(* IEC 61131-3 sources: AXOpen/src/components.siemens.identification/ctrl/src/IOLink, 6 files *)

(* ---- AxoIOLink_Device.st ---- *)
USING AXOpen.Components.Abstractions.Drives;
USING AXOpen.Timers;
USING Siemens.Simatic.S71500.DistributedIO;
USING System.Timer;

NAMESPACE AXOpen.Components.SIEM.Identification
    {S7.extern=ReadWrite}
    CLASS PUBLIC AxoIOLink_Device
        VAR PRIVATE
            statExecuteOld          :	BOOL    :=  FALSE;          //  Old value of 'execute' input for edge detection
            statDone                :	BOOL    :=  FALSE;          //  Static value for output 'done'
            statBusy                :	BOOL    :=  FALSE;          //  Static value for output 'busy'
            statError               :	BOOL    :=  FALSE;          //  Static value for output 'error'
            statStatus              :	WORD    :=  WORD#16#7000;	//  Static value for output 'status'
            statPollingPeriod       :	TIME    :=	T#100MS;        //	Static value for input 'pollingPeriod'
            statHwID                :	WORD    :=  WORD#0;         //  Static value for input 'hwID'
            statHwIDprevious        :	WORD    :=  WORD#0;         //  Static value for input 'hwID' from the previous execute
            statReadWrite           :	BOOL    :=  FALSE;          //  Static value for input 'readWrite'
            statCap                 :	UINT    :=  UINT#0;         //  Static value for input 'cap'
            statTimeout             :	TIME    :=	T#0MS;          //	Static value for input 'timeout'
            statLen                 :	UINT    :=  UINT#0;         //  Length of data to be written to device
            statSubfunctionStatus   :	DWORD   :=  DWORD#0;        //  Status of WRREC/RDREC or error code from IO-Link Master (%W1: IO-Link Master error, %W0: ISDU error)
            statFBErrorState        :	DINT    :=  DINT#0;         //	State in the state machine of the block where the error occurred
            statFBState             :	DINT    :=  DINT#0;         //	State in the state machine of the FB
            statEmptyDiagnostics    :	AxoIOLink_typeDiagnostics;  //  Empty diagnostics information (for initialization purposes only)
            instRdRec               :	ReadRecord;                 //  System function "read data record"
            instWrRec               :	WriteRecord;                //  System function "write data record"
            instPoll                :	Pulse;  		            //  poll rate read data record
            instMonitor             :	OnDelay;                    //  request monitoring time
            statRead                :	ARRAY[0..239] OF BYTE   := [BYTE#16#08,BYTE#16#0,BYTE#16#FE,BYTE#16#4A,236(BYTE#0)];             //  data area for reading data
            statWrite               :	ARRAY[0..239] OF BYTE   := [BYTE#16#08,BYTE#16#0,BYTE#16#FE,BYTE#16#4A,236(BYTE#0)];             //  data area for writing data
            statDiagnostics         :	AxoIOLink_typeDiagnostics;
            statReadLen             :	INT;

        END_VAR

        VAR CONSTANT
            MODE_READ                   :	BOOL    :=	FALSE;              //  Mode to read data
            MODE_WRITE                  :	BOOL    :=	TRUE;               //  Mode to write data
            MAX_PORT                    :	USINT   :=  USINT#63;           //  Max. possible port
            MAX_INDEX                   :	UINT    :=  UINT#32767;         //  Max. possible index
            INDEX_PORT_FUNC             :	UINT    :=  UINT#65535;         //  Index to address port functions
            MAX_SUBINDEX                :	USINT   :=  USINT#255;          //  Max. possible subindex
            MAX_DATA                    :	USINT	:=  USINT#232;          //  Max. size of data to be transferred
            UPPER_LIMIT                 :	DINT    :=  DINT#231;           //  Upper limit of data to be transferred
            FB_STATE_NO_PROCESSING      :	DINT    :=  DINT#0;             //  FB state: No processing
            FB_STATE_WRITE              :	DINT    :=  DINT#1;             //  FB state: Write data record
            FB_STATE_POLL               :	DINT    :=  DINT#2;             //  FB state: Wait and poll for response
            FB_STATE_READ_CAP           :	DINT    :=  DINT#3;             //  FB state: Read cap
            IOL_HEADER                  :	UINT    :=  UINT#65098;         //  Header IO-Link
            LEN_HEADER                  :	USINT   :=  USINT#8;            //  Length of header
            CONTROL_WRITE               :	BYTE    :=  BYTE#16#02;         //  Write data record
            CONTROL_READ                :	BYTE    :=  BYTE#16#03;         //  Read data record
            STATUS_EXECUTION_FINISHED   :	WORD    :=  WORD#16#0000;       //  Execution finished without errors
            STATUS_NO_CALL              :	WORD    :=  WORD#16#7000;       //  No job being currently processed
            STATUS_FIRST_CALL           :	WORD    :=  WORD#16#7001;       //  First call after incoming new job (rising edge 'execute')
            STATUS_SUBSEQUENT_CALL      :	WORD    :=  WORD#16#7002;       //  Subsequent call during active processing without further details
            SUB_STATUS_NO_ERROR         :	WORD    :=  WORD#16#0000;       //  No error occured in subfunction call
            ERR_WRONG_PORT              :	WORD    :=  WORD#16#8201;       //  Error: wrong port
            ERR_WRONG_INDEX             :	WORD    :=  WORD#16#8202;       //  Error: wrong index
            ERR_WRONG_SUBINDEX          :	WORD    :=  WORD#16#8203;       //  Error: wrong subindex
            ERR_WRONG_LENGTH            :	WORD    :=  WORD#16#8205;       //  Error: wrong length for write data record
            ERR_IO_LINK                 :	WORD    :=  WORD#16#8401;       //  Error: IO-Link master returned error code, see "diagnostics"
            ERR_INCONSISTENT_DATA       :	WORD    :=  WORD#16#8402;       //  Error: Read data record doesn't match request
            ERR_REQUEST_TIMEOUT         :	WORD    :=  WORD#16#8403;       //  Error: Request timed out
            ERR_UNDEFINED_STATE         :	WORD    :=  WORD#16#8600;       //  Error: due to an undefined state in state machine
            ERR_WRREC                   :	WORD    :=  WORD#16#8601;       //  Error: WRREC encountered an error, see "diagnostics"
            ERR_RDREC                   :	WORD    :=  WORD#16#8602;       //  Error: RDREC encountered an error, see "diagnostics"
            STATUS_MASK                 :	DWORD   :=  DWORD#16#00FF_FF00; //  Mask to filter error codes
            STATUS_RESOURCE_BUSY        :	DWORD   :=  DWORD#16#0080_C200; //  Status from WRREC/RDREC: Resource is busy
            INDEX_CAP_IOLINK            :	WORD    :=  WORD#16#B000;       //  Index of the data record for IOLM_Info. Only IO-Link-Masters with CAP=16#B000 support this call.
            CAP_LEGACY                  :	WORD    :=  WORD#16#00E3;       //  Siemens (old) Standard CAP: 227
            CAP_STANDARD                :	WORD    :=  WORD#16#B400;       //  IO-Link Standard CAP: 16#B400
            STATUS_RDREC_VALID          :	BYTE    :=  BYTE#16#00;         //  Status Code of RDREC in cased of no error occurs
            BITMASK_ERR_RDREC_B3        :	BYTE    :=  BYTE#16#DE;         //  Status Code of RDREC in case of an error when reading a data record
            BITMASK_ERR_RDREC_B2        :	BYTE    :=  BYTE#16#80;         //  Status Code of RDREC in case of an error when reading a data record - Error according to IEC 61158-6
            BITMASK_ERR_RDREC_B1        :	BYTE    :=  BYTE#16#B0;         //  Status Code of RDREC in case of an error when reading a data record - invalid index (cap)
        END_VAR

        METHOD PUBLIC Run
            VAR_INPUT
                execute         :	BOOL    :=  FALSE;                  //	Request to execute function
                hwID            :	WORD    :=  WORD#0;                 //	Hardware identifier of IO-Link master module or first sub module
                cap             :	INT     :=  INT#0;                  //	Client Access Point (CAP) 0xB400 or 0x00E3 (227)
                readWrite       :	BOOL    :=  FALSE;                  //	FALSE: read-mode, TRUE: write-mode
                port            :	INT     :=  INT#0;                  //  Port on IO-Link master module
                index           :	INT     :=  INT#0;                  //  Address parameter index (IO-Link device); 0..32767: IOL-D; 65535: port functions
                subindex        :	INT     :=  INT#0;                  //  Address parameter subindex (IO-Link device); 0: full record; 1-255: single parameter
                writeLen        :	INT     :=  INT#0;                  //  Length of writing data (net data); 1..232
                timeout         :	TIME    :=	T#20S;                  //	Time after which the request is aborted
                pollingPeriod   :	TIME    :=	T#100MS;                //	Time period of polling
                record	        :   REF_TO Array[*] OF BYTE;            //  Data area for reading/writing data (max. 232 byte)
                diagnostics     :	REF_TO  AxoIOLink_typeDiagnostics;	//  Diagnostics information of FB
            END_VAR

            VAR_OUTPUT
                done        :	BOOL;                                   //  TRUE: FB processing successfully completed
                busy        :	BOOL;                                   //  TRUE: FB is active and new output values can be expected.
                error       :	BOOL;                                   //  FALSE: No error / TRUE: An error occurred during the execution of the FB.
                status      :	WORD;                                   //  16#0000-16#7FFF: Status of the FB / 16#8000-16#FFFF: Error identification (see following table)
                readLen     :	INT;                                    //  Length of read data record (number of bytes)
            END_VAR

            VAR_TEMP
                tempExecute         :	BOOL;							//	Temporary value for input 'execute'
                tempHwID            :	WORD;							//	Temporary value for input 'hwID'
                tempPort            :	INT;							//	Temporary value for input 'port'
                tempIndex           :	INT;							//	Temporary value for input 'index'
                tempSubindex        :	INT;							//	Temporary value for input 'subindex'
                tempIndexCounter    :	DINT;							//	run tag for counting loops
                i                   :   INT;
            END_VAR

            IF record = NULL THEN
                // TODO some message
                RETURN;
            END_IF;

            IF diagnostics = NULL THEN
                // TODO some message
                RETURN;
            END_IF;

            //===============================================================================
            // Siemens / (c)Copyright 2023
            //-------------------------------------------------------------------------------
            // Title:            LIOLink_Device
            // Function:         Acyclically reads or writes data records from and to IO-Link devices
            // Library:          LIOLink
            // Author:           Siemens Industry Online Support
            // Tested with:      CPU 1513-1 PN FW 2.8
            // Engineering:      TIA Portal V16
            // Restrictions:     S7-1200/1500
            // Requirements:     --
            //-------------------------------------------------------------------------------
            // Change log table:
            // Version  | Date       | Expert in charge       | Changes applied
            //----------|------------|------------------------|------------------------------
            // 02.00.00 | 30.09.2013 | Online Support         | First release for TIA Portal V12 SP1 as IO_LINK_CALL
            // 02.01.00 | 14.03.2014 | Online Support         | Upgrade to TIA Portal V13
            //                                                | Upgrade of system function 'WRREC' from V1.0 to V1.1
            // 03.00.00 | 28.02.2015 | SUP Applications       | Upgrade to TIA Portal V13 SP1
            //                                                | Renamed FB to IO_LINK_DEVICE
            // 03.01.00 | 15.09.2015 | SUP Applications       | Change of #IOL_INDEX AND #Port lower boundry to 0 and improved behaviour when called in cyclic OBs with > 100 ms
            // 04.00.00 | 01.09.2020 | Online Support         | Implemented Programming styleguide for S7-1200/1500 and PLCopen
            //                                                | Renamed FB to LIOLink_Device
            // 05.00.00 | 28.02.2023 | SUP SPH                | Added Polling Time as predefined input
            //                                                | #record is changed to a variable array (Array[*])
            //                                                | Changed CAP as predefined variable, added functionality to automatically find CAP of IO-Link-Masters from SIEMENS
            //===============================================================================
            // TRIGGERING
            tempExecute := execute; // Work with temporary value / create process image

            IF (tempExecute = TRUE) AND (statExecuteOld = FALSE) // Check if FB is triggered
                AND (statStatus = STATUS_NO_CALL)
            THEN
                    // First call; initialize FB
                    statDone := FALSE;
                    statBusy := TRUE;
                    statError := FALSE;
                    statStatus := STATUS_FIRST_CALL;
                    statSubfunctionStatus := SUB_STATUS_NO_ERROR;
                    statFBErrorState := 0;
                    statDiagnostics := statEmptyDiagnostics;
                    statReadLen := 0;

                    // Initialize data area
                    statRead[0] := BYTE#16#0;
                    statRead[6] := BYTE#16#0;
                    statRead[5] := BYTE#16#0;
                    statRead[7] := BYTE#16#0;
                    tempIndexCounter := 0; // initialize loop counter
                    FOR tempIndexCounter := 0 TO UPPER_LIMIT + 8 DO
                        statWrite[tempIndexCounter] := BYTE#16#0;
                        statRead[tempIndexCounter] := BYTE#16#0;
                    END_FOR;

                    // Copy input variables to temporary variables
                    tempHwID := hwID;
                    statReadWrite := readWrite;
                    statTimeout := timeout;
                    statPollingPeriod := pollingPeriod;
                    tempPort := port;
                    tempIndex := index;
                    tempSubindex := subindex;

                    // setup call header
                    statWrite[0] := TO_BYTE(tempPort);
                    // setup IOL header
                    statWrite[6] := TO_BYTE(tempIndex);
                    statWrite[5] := TO_BYTE(SHR(TO_WORD(tempIndex), UINT#8));
                    statWrite[7] := TO_BYTE(tempSubindex);

                    // BODY (data max. 232 Byte, Array 0..231 of Byte)
                    IF statReadWrite = MODE_WRITE THEN // Write data record requested, copy data from "record"
                        statWrite[4] := CONTROL_WRITE;
                        statLen := TO_UINT(writeLen) + LEN_HEADER; // data length header + data = IO-Link write data record
                        // copy "record" to working area
                        FOR tempIndexCounter := 8 TO writeLen - 7 DO
                            statWrite[tempIndexCounter] := record^[tempIndexCounter];
                        END_FOR;
                    ELSE // Read data record requested
                        // Empty record array
                        FOR i := 0 TO MAX_DATA DO
                            record^[0] := BYTE#0;
                        END_FOR;
                        statWrite[4] := CONTROL_READ;
                        statLen := LEN_HEADER; // data length only header = IO-Link read data record
                    END_IF;

                    // Check parameters
                    IF (tempPort < 0) OR (tempPort > MAX_PORT) THEN
                        statStatus := ERR_WRONG_PORT;
                    ELSIF (tempIndex < 0) OR (TO_UINT(tempIndex) > MAX_INDEX AND TO_UINT(tempIndex) <> INDEX_PORT_FUNC) THEN
                        statStatus := ERR_WRONG_INDEX;
                    ELSIF (tempSubindex < 0) OR (tempSubindex > MAX_SUBINDEX) THEN
                        statStatus := ERR_WRONG_SUBINDEX;
                    ELSIF statReadWrite = MODE_WRITE AND (writeLen < 1 OR writeLen > MAX_DATA) THEN
                        statStatus := ERR_WRONG_LENGTH;
                    END_IF;
                    //save the hwID from the previous execute
                    statHwIDprevious := statHwID;

                    IF statStatus = STATUS_FIRST_CALL THEN // Parameters OK
                        IF cap <> 0 THEN
                            statCap := TO_UINT(cap);
                            statFBState := FB_STATE_WRITE;
                        ELSIF (statCap <> TO_UINT(CAP_STANDARD) AND statCap <> TO_UINT(CAP_LEGACY)) OR (statHwIDprevious <> tempHwID) THEN // check if new device is connected => hwID changed
                            statFBState := FB_STATE_READ_CAP;
                        ELSE
                            statFBState := FB_STATE_WRITE;
                        END_IF;
                    END_IF;
                    // save current hwID
                    statHwID := tempHwID;

            ELSIF (statStatus = STATUS_FIRST_CALL) THEN
                statStatus := STATUS_SUBSEQUENT_CALL;
            END_IF;

            // Edge detection 'execute' input
            statExecuteOld := tempExecute;

            // STATE_MACHINE
            CASE statFBState OF
                FB_STATE_NO_PROCESSING:
                        ; // No processing active

                FB_STATE_READ_CAP:
                        // To find out CAP of IO-Link Master, data record with Index 16#B000 is read. If this reading was successful
                        // then CAP is 16#B400 (based on IO-Link Standard). If the reading was not successful and the status of RDREC
                        // is 16#DE80_B0xx, then CAP is 16#00E3 (227, based on Siemens Old Standard for IO-Link Masters).

                        instRdRec(record := statRead);

                        IF (instRdRec.BUSY = FALSE) THEN
                            IF (instRdRec.VALID = FALSE) AND (instRdRec.ERROR = FALSE) THEN
                                IF instRdRec.request = FALSE THEN
                                    // call read record with Index 16#B000
                                    instRdRec.request := true;
                                    instRdRec.ID := statHwID;
                                    instRdRec.INDEX := TO_UINT(INDEX_CAP_IOLINK);
                                    instRdRec.maxLength := UINT#0;
                                    statFBState := FB_STATE_READ_CAP;
                                END_IF;
                            ELSIF instRdRec.VALID = TRUE THEN
                                instRdRec.request := FALSE;
                                // if status of RDREC is valid then CAP is 16#B400 (CAP_STANDARD)
                                IF instRdRec.STATUS.%B3 = STATUS_RDREC_VALID THEN
                                    statCap := TO_UINT(CAP_STANDARD);
                                END_IF;
                                statFBState := FB_STATE_WRITE;
                            ELSE
                                // if RDREC is in error state and Status is 16#DE80_B0xx then CAP is 227 (CAP_Legacy)
                                IF (instRdRec.STATUS.%B3 = BITMASK_ERR_RDREC_B3) AND (instRdRec.STATUS.%B2 = BITMASK_ERR_RDREC_B2) AND (instRdRec.STATUS.%B1 = BITMASK_ERR_RDREC_B1) THEN
                                    statCap := TO_UINT(CAP_LEGACY);
                                    statFBState := FB_STATE_WRITE;
                                ELSE
                                    statStatus := ERR_RDREC;
                                    statSubfunctionStatus := instRdRec.STATUS;
                                    statCap := UINT#0; //clear CAP if an error occurs
                                END_IF;
                            END_IF;
                        ELSE
                            instRdRec.request := FALSE;
                            IF instRdRec.ERROR = TRUE THEN
                                statStatus := ERR_RDREC;
                                statSubfunctionStatus := instRdRec.STATUS;
                                statCap := UINT#0; //clear CAP if an error occurs
                            END_IF;
                        END_IF;

                        instRdRec(RECORD := statRead);

                FB_STATE_WRITE:
                        // To read data records, the IO-Link master modules needs to know which port is required. Therefore it is necessary
                        // to send at first a request via write data record (header, 8 byte). As response the IO-Link master module will
                        // send the required data record.

                        instWrRec(request := TRUE,
                                   id := statHwID,
                                   index := statCap,
                                   length := statLen,
                                   record := statWrite);

                        IF instWrRec.ERROR THEN
                            IF (instWrRec.STATUS AND STATUS_MASK) = STATUS_RESOURCE_BUSY THEN
                                instWrRec(request := FALSE,record := statWrite); // Reset request
                            ELSE
                                statStatus := ERR_WRREC;
                                statSubfunctionStatus := instWrRec.STATUS;
                                statFBErrorState := statFBState;
                            END_IF;
                        ELSIF instWrRec.DONE = TRUE THEN
                            instWrRec(request := FALSE,record := statWrite); // Reset requeset

                            statFBState := FB_STATE_POLL;
                        END_IF;

                FB_STATE_POLL: // wait and poll for response
                        instPoll(signal := TRUE,
                                  duration := statPollingPeriod);

                        // read data record on falling edge
                        instRdRec(request := NOT instPoll.output,
                                   id := statHwID,
                                   index := statCap,
                                   maxLength := UINT#0, // read all data available,
                                   record := statRead);

                        IF instRdRec.ERROR = TRUE THEN
                            IF (instRdRec.STATUS AND STATUS_MASK) = STATUS_RESOURCE_BUSY THEN
                                // Reset requests and try again
                                instPoll(signal := FALSE,duration := statPollingPeriod);

                                instRdRec(request := FALSE,record := statRead);
                            ELSE
                                statStatus := ERR_RDREC;
                                statSubfunctionStatus := instRdRec.STATUS;
                                statFBErrorState := statFBState;
                            END_IF;
                        ELSIF instRdRec.VALID THEN
                            IF // check the response wether it matches the request (compare PORT, INDEX and SUBINDEX)
                                (statWrite[0] <> statRead[0])
                                OR (statWrite[5] <> statRead[5])
                                OR (statWrite[6] <> statRead[6])
                                OR (statWrite[7] <> statRead[7])
                            THEN // read data record doesn't match the request
                                statStatus := ERR_INCONSISTENT_DATA;  // output status no consistent data
                            ELSIF statRead[4] = BYTE#16#80 THEN // check the response for IO-Link errors
                                // State 0x80 = IOL_CALL_RES PDU shows IO-Link error detect
                                statStatus := ERR_IO_LINK;
                                statSubfunctionStatus.%B3 := statRead[8]; // IO-Link master error code
                                statSubfunctionStatus.%B2 := statRead[9]; // IO-Link master error code
                                statSubfunctionStatus.%B1 := statRead[10]; // ISDU error code
                                statSubfunctionStatus.%B0 := statRead[11]; // ISDU additional code
                                statFBErrorState := statFBState;
                            ELSE // read data is valid
                                IF statReadWrite = MODE_READ THEN
                                    statReadLen := TO_INT(instRdRec.length - LEN_HEADER);
                                    // only data will be output
                                    FOR tempIndexCounter := 0 TO TO_INT(instRdRec.length - TO_UINT(LEN_HEADER) - UINT#1) DO
                                        record^[tempIndexCounter] := statRead[tempIndexCounter + DINT#8];
                                    END_FOR;
                                END_IF;

                                // Reset requests
                                instRdRec(request := FALSE,record := statRead);

                                instPoll(signal := FALSE,duration := statPollingPeriod);

                                statStatus := STATUS_EXECUTION_FINISHED;  // request finished
                            END_IF;
                        END_IF;

                ELSE // Undefined state in state machine reached
                        statStatus := ERR_UNDEFINED_STATE;
            END_CASE;

            //  MONITORING
            instMonitor(signal := statBusy,duration := statTimeout);

            IF instMonitor.output THEN
                statStatus := ERR_REQUEST_TIMEOUT; // request time out
            END_IF;

            // OUTPUTS
            // Write outputs
            IF (statStatus = STATUS_EXECUTION_FINISHED) AND (statDone = FALSE) THEN // Execution finished without errors, available only for one cycle
                    statDone := TRUE;
                    statBusy := FALSE;
                    statError := FALSE;
                    // execution aborted --> set state no processing
                    statFBState := FB_STATE_NO_PROCESSING;

            ELSIF (statStatus.%X15 = TRUE) AND (statError = FALSE) THEN // Error occurred (statStatus is 16#8000 to 16#FFFF), Error status is true only for one cycle (the second last cycle)
                    statDone := FALSE;
                    statBusy := FALSE;
                    statError := TRUE;
                    statCap := UINT#0; //Reset statcap, if error occurs, get cap has to be performed again
                    // Write diagnostics
                    statDiagnostics.status := statStatus;
                    statDiagnostics.subfunctionStatus := statSubfunctionStatus;
                    statDiagnostics.stateNumber := statFBErrorState;
                    // Call instructions with FALSE to be ready for next job
                    instWrRec(request := FALSE,record := statWrite);

                    instRdRec(request := FALSE,record := statRead);

                    instPoll(signal := FALSE,duration := statPollingPeriod);

                    // execution aborted --> set state no processing
                    statFBState := FB_STATE_NO_PROCESSING;

            ELSIF (tempExecute = FALSE) AND ((statDone = TRUE) OR (statError = TRUE)) THEN // Reset outputs, Last cycle
                    statDone := FALSE;
                    statBusy := FALSE;
                    statError := FALSE;
                    statStatus := STATUS_NO_CALL;
                    statReadLen := 0;
            END_IF;

                done := statDone;
                busy := statBusy;
                error := statError;
                status := statStatus;
                readLen := statReadLen;
                diagnostics^ := statDiagnostics;
                //ENO := NOT statError;
        END_METHOD
    END_CLASS
END_NAMESPACE

(* ---- AxoIOLink_RF200.st ---- *)
USING AXOpen.Components.Abstractions.Drives;
USING AXOpen.Timers;
USING Siemens.Simatic.S71500.DistributedIO;
USING System.Timer;
USING System.Strings;
USING System.Serialization;

NAMESPACE AXOpen.Components.SIEM.Identification
    {S7.extern=ReadWrite}
    CLASS PUBLIC AxoIOLink_RF200
        VAR PRIVATE
            instDevice                  :	AxoIOLink_Device;                       //  Acyclically reads or writes data records from and to IO-Link devices
            statRecordParam_index       :   ARRAY[0..HIGHEST_REQUEST_NUMBER] OF INT :=  [0,INDEX_DIRECT_PARAM1,0,0,0,0,0,0,0,INDEX_EVENT_HISTORY,INDEX_VENDOR_NAME,INDEX_VENDOR_TEXT,INDEX_PRODUCT_NAME,INDEX_PRODUCT_ID,20,21,22,INDEX_FIRMWARE_REVISION,INDEX_APP_SPECIFIC_NAME,INDEX_ERROR_COUNT,0,0,INDEX_TAG_STATUS,INDEX_READER_STATUS,INDEX_UID_HISTORY,0,0,0,0];  //  Data set index
            statRecordParam_subindex    :	ARRAY[0..HIGHEST_REQUEST_NUMBER] OF INT :=  [29(0)];    //  Data set subindex
            statRecordParam_length      :	ARRAY[0..HIGHEST_REQUEST_NUMBER] OF INT :=  [0,LENGTH_DIRECT_PARAM1,0,0,0,0,0,0,0,LENGTH_EVENT_HISTORY,LENGTH_VENDOR_NAME,LENGTH_VENDOR_TEXT,LENGTH_PRODUCT_NAME,LENGTH_PRODUCT_ID,0,0,0,LENGTH_FIRMWARE_REVISION,LENGTH_APP_SPECIFIC_NAME,LENGTH_ERROR_COUNT,0,0,LENGTH_TAG_STATUS,LENGTH_READER_STATUS,LENGTH_UID_HISTORY,0,0,0,0]; //  Data set length
            statRecord                  :	ARRAY[0..UPPER_BOUND_RECORD] OF BYTE;   //  Record buffer
            statIndex                   :	INT     :=  INT#0;                      //	Requested index
            statSubindex                :	INT     :=  INT#0;                      //	Requested subindex
            statRecordLen               :	INT     :=  INT#0;                      //	Length of record to be written
            statHwID                    :	WORD    :=  WORD#0;                     //  Static value for input 'hwID'
            statCap                     :	INT     :=  INT#0;                      //  Static value for input 'cap'
            statReadWrite               :	BOOL    :=  FALSE;                      //  Static value for input 'readWrite'
            statPort                    :	INT     :=  INT#0;                      //  Static value for input 'port'
            statPollingPeriod           :	Time	:=  T#0ms;                      //  Static value for input 'pollingPeriod'
            statDirectParameter1        :	BOOL    :=  FALSE;                      //  Static value for input 'directParameter1'
            statSystemCommand           :	BOOL    :=  FALSE;                      //  Static value for input 'systemCommands'
            statDeviceAccessLocks       :	BOOL    :=  FALSE;                      //  Static value for input 'deviceAccessLocks'
            statVendorName              :	BOOL    :=  FALSE;                      //  Static value for input 'vendorName'
            statVendorText              :	BOOL    :=  FALSE;                      //  Static value for input 'vendorText'
            statProductName             :	BOOL    :=  FALSE;                      //  Static value for input 'productName'
            statProductID               :	BOOL    :=  FALSE;                      //  Static value for input 'productID'
            statProductText             :	BOOL    :=  FALSE;                      //  Static value for input 'productText'
            statSerialNumber            :	BOOL    :=  FALSE;                      //  Static value for input 'serialNumber'
            statHwRevision              :	BOOL    :=  FALSE;                      //  Static value for input 'hwRevision'
            statFwRevision              :	BOOL    :=  FALSE;                      //  Static value for input 'fwRevision'
            statAppSpecificName         :	BOOL    :=  FALSE;                      //  Static value for input 'appSpecificName'
            statErrorCount              :	BOOL    :=  FALSE;                      //  Static value for input 'errorCount'
            statDeviceStatus            :	BOOL    :=  FALSE;                      //  Static value for input 'deviceStatus'
            statDeviceStatusDetailed    :	BOOL    :=  FALSE;                      //  Static value for input 'deviceStatusDetailed'
            statProcessIn               :	BOOL    :=  FALSE;                      //  Static value for input 'processIn'
            statProcessOut              :	BOOL    :=  FALSE;                      //  Static value for input 'processOut'
            statParameters              :	BOOL    :=  FALSE;                      //  Static value for input 'parameters'
            statEventHistory            :	BOOL    :=  FALSE;                      //  Static value for input 'eventHistory'
            statReaderStatus            :	BOOL    :=  FALSE;                      //  Static value for input 'readerStatus'
            statTagStatus               :	BOOL    :=  FALSE;                      //  Static value for input 'tagStatus'
            statUidHistory              :	BOOL    :=  FALSE;                      //  Static value for input 'uidHistory'
            statRequest                 :	INT     :=  INT#0;                      //  Case of request (data set)
            statDoneOld                 :	BOOL    :=  FALSE;                      //  Last cycle's value of instDevice.done
            instDevice_done             :	BOOL    :=  FALSE;
            instDevice_busy             :	BOOL    :=  FALSE;
            instDevice_error            :	BOOL    :=  FALSE;
            instDevice_status           :	WORD    :=  WORD#0;
            instDevice_readLen          :	INT     :=  INT#0;
            instDevice_diagnostics      :   AxoIOLink_typeDiagnostics;
        END_VAR

        VAR CONSTANT
            UPPER_BOUND_RECORD              :	INT     :=  INT#231;        //				        Upper Bound of record buffer
            HIGHEST_REQUEST_NUMBER          :	INT     :=  INT#28;         //				        Highest available request number
            UPPER_BOUND_PARAMETER_PAGE0     :	INT     :=  INT#15;         //				        Upper Bound of Parameter Page 0 auxiliary field
            UPPER_BOUND_PARAMETERS          :	INT     :=  INT#7;          //				        Upper Bound of Parameters auxiliary field
            UPPER_BOUND_EVENT_HISTORY       :	INT     :=  INT#19;         //				        Upper Bound of Event History auxiliary field
            UPPER_BOUND_READER_STATUS       :	INT     :=  INT#17;         //				        Upper Bound of Reader Status auxiliary field
            UPPER_BOUND_TAG_STATUS          :	INT     :=  INT#15;         //				        Upper Bound of Tag Status auxiliary field
            UPPER_BOUND_UID_HISTORY         :	INT     :=  INT#39;         //				        Upper Bound of UID History auxiliary field
            MODE_READ                       :	BOOL    :=	FALSE;          //						Mode to read data
            MODE_WRITE                      :	BOOL    :=	TRUE;           //						Mode to write data
            STATUS_IDLE                     :	WORD    :=  WORD#16#7000;   //						Status: Idle
            STATUS_EXECUTION_FINISHED       :	WORD    :=  WORD#16#0000;   //						Execution finished without errors
            ERR_INCONSISTENT_DATA           :	WORD    :=  WORD#16#8402;   //						Error: Read data record doesn't match request
            INDEX_DIRECT_PARAM1             :	INT     :=  INT#0;          //						Record Index
            INDEX_SYSTEM_COMMAND            :	INT     :=  INT#2;          //						Record Index
            INDEX_ACCESS_LOCKS              :	INT     :=  INT#12;         //						Record Index
            INDEX_EVENT_HISTORY             :	INT     :=  INT#74;         //						Record Index
            INDEX_VENDOR_NAME               :	INT     :=  INT#16;         //						Record Index
            INDEX_VENDOR_TEXT               :	INT     :=  INT#17;         //						Record Index
            INDEX_PRODUCT_NAME              :	INT     :=  INT#18;         //						Record Index
            INDEX_PRODUCT_ID                :	INT     :=  INT#19;         //						Record Index
            INDEX_PRODUCT_TEXT              :	INT     :=  INT#20;         //						Record Index
            INDEX_SERIAL_NUMBER             :	INT     :=  INT#21;         //						Record Index
            INDEX_HARDWARE_REVISION         :	INT     :=  INT#22;         //						Record Index
            INDEX_FIRMWARE_REVISION         :	INT     :=  INT#23;         //						Record Index
            INDEX_APP_SPECIFIC_NAME         :	INT     :=  INT#24;         //						Record Index
            INDEX_ERROR_COUNT               :	INT     :=  INT#32;         //						Record Index
            INDEX_DEVICE_STATUS             :	INT     :=  INT#36;         //						Record Index
            INDEX_DETAILED_STATUS           :	INT     :=  INT#37;         //						Record Index
            INDEX_PII                       :	INT     :=  INT#40;         //						Record Index
            INDEX_PIQ                       :	INT     :=  INT#41;         //						Record Index
            INDEX_PARAMETERS                :	INT     :=  INT#64;         //						Record Index
            INDEX_TAG_STATUS                :	INT     :=  INT#91;         //						Record Index
            INDEX_READER_STATUS             :	INT     :=  INT#90;         //						Record Index
            INDEX_UID_HISTORY               :	INT     :=  INT#92;         //						Record Index
            LENGTH_DIRECT_PARAM1            :	INT     :=  INT#16;         //						Record Length
            LENGTH_SYSTEM_COMMAND           :	INT     :=  INT#1;          //						Record Length
            LENGTH_ACCESS_LOCKS             :	INT     :=  INT#2;          //						Record Length
            LENGTH_EVENT_HISTORY            :	INT     :=  INT#20;         //						Record Length
            LENGTH_VENDOR_NAME              :	INT     :=  INT#12;         //						Record Length
            LENGTH_VENDOR_TEXT              :	INT     :=  INT#12;         //						Record Length
            LENGTH_PRODUCT_NAME             :	INT     :=  INT#24;         //						Record Length
            LENGTH_PRODUCT_ID               :	INT     :=  INT#16;         //						Record Length
            LENGTH_PRODUCT_TEXT             :	INT     :=  INT#64;         //						Record Length
            LENGTH_SERIAL_NUMBER            :	INT     :=  INT#12;         //						Record Length
            LENGTH_HARDWARE_REVISION        :	INT     :=  INT#12;         //						Record Length
            LENGTH_FIRMWARE_REVISION        :	INT     :=  INT#12;         //						Record Length
            LENGTH_APP_SPECIFIC_NAME        :	INT     :=  INT#32;         //						Record Length
            LENGTH_ERROR_COUNT              :	INT     :=  INT#2;          //						Record Length
            LENGTH_DEVICE_STATUS            :	INT     :=  INT#1;          //						Record Length
            LENGTH_DETAILED_STATUS          :	INT     :=  INT#1;          //						Record Length
            LENGTH_PII                      :	INT     :=  INT#8;          //						Record Length
            LENGTH_PIQ                      :	INT     :=  INT#8;          //						Record Length
            LENGTH_PARAMETERS               :	INT     :=  INT#8;          //						Record Length
            LENGTH_TAG_STATUS               :	INT     :=  INT#15;         //						Record Length
            LENGTH_READER_STATUS            :	INT     :=  INT#18;         //						Record Length
            LENGTH_UID_HISTORY              :	INT     :=  INT#40;         //						Record Length
            EMPTY_CHAR                      :	CHAR    :=  CHAR#'$00';     //						Default empty chat to fill empty field entries
            DEVICE_TIMEOUT                  :	TIME    :=	T#20S;          //						Timeout value for the IO-Link Device Instance

        END_VAR

        METHOD PUBLIC Run
            VAR_INPUT
                execute                 :	BOOL    :=  FALSE;                  //  Request job (on rising edge)
                hwID                    :	WORD    :=  WORD#0;                 //  Hardware identifier of IO-Link master module or first sub module
                cap                     :	INT     :=  INT#0;                  //  Client Access Point (CAP) 0xB400 or 0x00E3 (227)
                readWrite               :	BOOL    :=  FALSE;                  //  Read and write access to IO-Link device 0: Read, 1:Write
                port                    :	INT     :=  INT#0;                  //  Port of device on the IO-Link Master
                pollingPeriod           :	TIME    :=  T#100MS;                //	Time period of polling
                directParameter1        :	BOOL    :=  FALSE;                  //  Read parameter page 1
                systemCommand           :	BOOL    :=  FALSE;                  //  Read system commands
                deviceAccessLocks       :	BOOL    :=  FALSE;                  //  Read device access locks
                vendorName              :	BOOL    :=  FALSE;                  //  Read manufacturer name
                vendorText              :	BOOL    :=  FALSE;                  //  Read manufacturer text
                productName             :	BOOL    :=  FALSE;                  //  Read product name
                productID               :	BOOL    :=  FALSE;                  //  Read product ID
                productText             :	BOOL    :=  FALSE;                  //  Read product text
                serialNumber            :	BOOL    :=  FALSE;                  //  Read serial number
                hwRevision              :	BOOL    :=  FALSE;                  //  Read hardware revision
                fwRevision              :	BOOL    :=  FALSE;                  //  Read firmware revision
                appSpecificName         :	BOOL    :=  FALSE;                  //  Read/Write application specific name
                errorCount              :	BOOL    :=  FALSE;                  //  Read error count
                deviceStatus            :	BOOL    :=  FALSE;                  //  Read device status
                deviceStatusDetailed    :	BOOL    :=  FALSE;                  //  Read device status detailed
                processIn               :	BOOL    :=  FALSE;                  //  Read process data IN
                processOut              :	BOOL    :=  FALSE;                  //  Read process data OUT
                parameters              :	BOOL    :=  FALSE;                  //  Read parameters
                eventHistory            :	BOOL    :=  FALSE;                  //  Read event history
                readerStatus            :	BOOL    :=  FALSE;                  //  Read status of reader
                tagStatus               :	BOOL    :=  FALSE;                  //  Reag tag status
                uidHistory              :	BOOL    :=  FALSE;                  //  Read UID history
                diagnostics	            :   REF_TO  AxoIOLink_typeDiagnostics;  //  IO-Link error status
                data                    :   REF_TO	AxoIOLink_RF200_typeAll;    //  Device data buffer

            END_VAR

            VAR_OUTPUT
                done    :	BOOL;       //  FALSE: data invalid, TRUE: data valid
                busy    :	BOOL;       //  FALSE: job done, TRUE: job in progress
                error   :	BOOL;       //  FALSE: no error, TRUE: error
                status  :	WORD;       //  DP/PN IO error status

            END_VAR

            VAR_TEMP
                tempIndex                   :	UINT;								            //  Loop index
                tempLen                     :	UINT;								            //  Auxiliary tag Length
                tempRetValSerialize         :	INT;								            //  Auxiliary tag for Serialize RetVal
                tempRetValDeserialize       :	INT;								            //  Auxiliary tag for Deserialize RetVal
                tempPosSerialize            :	DINT;								            //  Auxiliary tag for Serialize POS
                tempPosDeserialize          :	DINT;								            //  Auxiliary tag for Deserialize POS Output
                tempFieldParameterPage0     :	ARRAY[0..UPPER_BOUND_PARAMETER_PAGE0] OF BYTE;  //	Auxiliary tag for Parameter Page 0 record conversion
                tempFieldParameters         :	ARRAY[0..UPPER_BOUND_PARAMETERS] OF BYTE;       //	Auxiliary tag for Parameters record conversion
                tempFieldEventHistory       :	ARRAY[0..UPPER_BOUND_EVENT_HISTORY] OF BYTE;    //	Auxiliary tag for EventHistory record conversion
                tempFieldReaderStatus       :	ARRAY[0..UPPER_BOUND_READER_STATUS] OF BYTE;    //	Auxiliary tag for Reader Status record conversion
                tempFieldTagStatus          :	ARRAY[0..UPPER_BOUND_TAG_STATUS] OF BYTE;       //	Auxiliary tag for Tag Status record conversion
                tempFieldUIDHistory         :	ARRAY[0..UPPER_BOUND_UID_HISTORY] OF BYTE;      //	Auxiliary tag for UID History record conversion
                tempInternalError           :	BOOL;                                           //  Auxiliary tag to collect serialize and Deserialize issues
                tempData256                 :   ARRAY[0..255] OF BYTE;
            END_VAR

            IF data = NULL THEN
                // TODO some message
                RETURN;
            END_IF;

            IF diagnostics = NULL THEN
                // TODO some message
                RETURN;
            END_IF;

            // INFO HEADER
            //===============================================================================
            // Siemens / (c)Copyright 2023
            //-------------------------------------------------------------------------------
            // Title:            LIOLink_RF200
            // Function:         Capsule block to communicate with SIMATIC RF200 Readers
            // Library:          LIOLink
            // Author:           Siemens Industry Online Support
            // Tested with:      CPU 1513-1 PN FW 2.8
            // Engineering:      TIA Portal V16
            // Restrictions:     --
            // Requirements:     --
            //-------------------------------------------------------------------------------
            // Change log table:
            // Version  | Date       | Expert in charge       | Changes applied
            //----------|------------|------------------------|------------------------------
            // 01.00.00 | 11.04.2014 | Online Support         | First release
            // 02.00.00 | 30.03.2015 | Online Support         | Upgrade to TIA Portal V13 SP1, use function IO_LINK_DEVICE, only one function for S7-1200 and 1500
            // 02.01.00 | 23.10.2015 | Online Support         | Update to IO_LINK_DEVICE Version 3.1
            // 03.00.00 | 01.09.2020 | Online Support         | Rewrote block for FB "LIOLink_Device" V4.0.0
            // 03.01.00 | 25.10.2022 | SUP SPH                | Optimized and function extension
            //===============================================================================

            // INIT
            IF (execute = TRUE AND instDevice_status = STATUS_IDLE) THEN

                // Inputs
                    //save inputs
                    statHwID := hwID;
                    statCap := cap;
                    statReadWrite := readWrite;
                    statPort := port;
                    statPollingPeriod := pollingPeriod;
                    statDirectParameter1 := directParameter1;
                    statSystemCommand := systemCommand;
                    statDeviceAccessLocks := deviceAccessLocks;
                    statVendorName := vendorName;
                    statVendorText := vendorText;
                    statProductName := productName;
                    statProductID := productID;
                    statProductText := productText;
                    statSerialNumber := serialNumber;
                    statHwRevision := hwRevision;
                    statFwRevision := fwRevision;
                    statAppSpecificName := appSpecificName;
                    statErrorCount := errorCount;
                    statDeviceStatus := deviceStatus;
                    statDeviceStatusDetailed := deviceStatusDetailed;
                    statProcessIn := processIn;
                    statProcessOut := processOut;
                    statParameters := parameters;
                    statEventHistory := eventHistory;
                    statReaderStatus := readerStatus;
                    statTagStatus := tagStatus;
                    statUidHistory := uidHistory;

                // Request selector
                    //set Index and RecordLen based on the request
                    IF statDirectParameter1 THEN
                        statIndex := INDEX_DIRECT_PARAM1;
                        statRecordLen := LENGTH_DIRECT_PARAM1;
                    ELSIF statSystemCommand THEN
                        statIndex := INDEX_SYSTEM_COMMAND;
                        statRecordLen := LENGTH_SYSTEM_COMMAND;
                    ELSIF statDeviceAccessLocks THEN
                        statIndex := INDEX_ACCESS_LOCKS;
                        statRecordLen := LENGTH_ACCESS_LOCKS;
                    ELSIF statVendorName THEN
                        statIndex := INDEX_VENDOR_NAME;
                        statRecordLen := LENGTH_VENDOR_NAME;
                    ELSIF statVendorText THEN
                        statIndex := INDEX_VENDOR_TEXT;
                        statRecordLen := LENGTH_VENDOR_TEXT;
                    ELSIF statProductName THEN
                        statIndex := INDEX_PRODUCT_NAME;
                        statRecordLen := LENGTH_PRODUCT_NAME;
                    ELSIF statProductID THEN
                        statIndex := INDEX_PRODUCT_ID;
                        statRecordLen := LENGTH_PRODUCT_ID;
                    ELSIF statProductText THEN
                        statIndex := INDEX_PRODUCT_TEXT;
                        statRecordLen := LENGTH_PRODUCT_TEXT;
                    ELSIF statSerialNumber THEN
                        statIndex := INDEX_SERIAL_NUMBER;
                        statRecordLen := LENGTH_SERIAL_NUMBER;
                    ELSIF statHwRevision THEN
                        statIndex := INDEX_HARDWARE_REVISION;
                        statRecordLen := LENGTH_HARDWARE_REVISION;
                    ELSIF statFwRevision THEN
                        statIndex := INDEX_FIRMWARE_REVISION;
                        statRecordLen := LENGTH_FIRMWARE_REVISION;
                    ELSIF statAppSpecificName THEN
                        statIndex := INDEX_APP_SPECIFIC_NAME;
                        statRecordLen := LENGTH_APP_SPECIFIC_NAME;
                    ELSIF statErrorCount THEN
                        statIndex := INDEX_ERROR_COUNT;
                        statRecordLen := LENGTH_ERROR_COUNT;
                    ELSIF statDeviceStatus THEN
                        statIndex := INDEX_DEVICE_STATUS;
                        statRecordLen := LENGTH_DEVICE_STATUS;
                    ELSIF statDeviceStatusDetailed THEN
                        statIndex := INDEX_DETAILED_STATUS;
                        statRecordLen := LENGTH_DETAILED_STATUS;
                    ELSIF statProcessIn THEN
                        statIndex := INDEX_PII;
                        statRecordLen := LENGTH_PII;
                    ELSIF statProcessOut THEN
                        statIndex := INDEX_PIQ;
                        statRecordLen := LENGTH_PIQ;
                    ELSIF statParameters THEN
                        statIndex := INDEX_PARAMETERS;
                        statRecordLen := LENGTH_PARAMETERS;
                    ELSIF statEventHistory THEN
                        statIndex := INDEX_EVENT_HISTORY;
                        statRecordLen := LENGTH_EVENT_HISTORY;
                    ELSIF statReaderStatus THEN
                        statIndex := INDEX_READER_STATUS;
                        statRecordLen := LENGTH_READER_STATUS;
                    ELSIF statTagStatus THEN
                        statIndex := INDEX_TAG_STATUS;
                        statRecordLen := LENGTH_TAG_STATUS;
                    ELSIF statUidHistory THEN
                        statIndex := INDEX_UID_HISTORY;
                        statRecordLen := LENGTH_UID_HISTORY;
                    ELSE
                        RETURN;
                    END_IF;

                IF statReadWrite = MODE_WRITE THEN
                    //prepare statRecord in case of a writing request
                    // write
                        IF statSystemCommand THEN
                            statRecord[0] := data^.systemCommand;

                        ELSIF statDeviceAccessLocks THEN
                            statRecord[0] := data^.deviceAccessLocks.%B0;
                            statRecord[1] := data^.deviceAccessLocks.%B1;

                        ELSIF statAppSpecificName THEN
                            tempLen :=  TO_UINT(LengthOf(data^.appSpecificName));
                            Serialize(UINT#0,data^.appSpecificName,tempData256);
                            FOR tempIndex := UINT#0 TO tempLen - UINT#1 DO
                                statRecord[tempIndex] :=   tempData256[tempIndex + UINT#1];
                            END_FOR;
                        ELSIF statParameters THEN
                                      statRecord[0] := data^.parameters.eventMessage;
                                      statRecord[1] := data^.parameters.operatingMode;
                                      statRecord[2] := data^.parameters.readyDelay;
                                      statRecord[3] := data^.parameters.dataHoldingTime;
                                      statRecord[4] := data^.parameters.rfParameters;
                                      statRecord[5] := data^.parameters.modulation;
                                      statRecord[6] := data^.parameters.subcarrier;
                                      statRecord[7] := data^.parameters.dataTransfer;

                            // Fill remaining characters with null
                            FOR tempIndex := UINT#8 TO TO_UINT(statRecordLen - 1) DO
                                statRecord[tempIndex] := TO_BYTE(EMPTY_CHAR);
                            END_FOR;
                        ELSE // all other data sets are read only
                            ;
                        END_IF;
                        tempInternalError := tempRetValSerialize <> TO_INT(STATUS_EXECUTION_FINISHED);
                END_IF;
            END_IF;

            //CALL
            //IOL-Call -> Request to read/write from an IO-Link-Device
            instDevice.Run(execute      := execute,
                        hwID            := statHwID,
                        cap             := statCap,
                        readWrite       := statReadWrite,
                        port            := statPort,
                        pollingPeriod   := statPollingPeriod,
                        index           := statIndex,
                        subindex        := statSubindex,
                        writeLen        := statRecordLen,
                        timeout         := DEVICE_TIMEOUT,
                        record          := REF(statRecord),
                        diagnostics     :=  REF(instDevice_diagnostics),
                        done            =>  instDevice_done    ,
                        busy            =>  instDevice_busy    ,
                        error           =>  instDevice_error   ,
                        status          =>  instDevice_status  ,
                        readLen         =>  instDevice_readLen );

            // READ
            // Copy data if available and valid
            IF instDevice_done = TRUE AND statDoneOld = FALSE AND statReadWrite = MODE_READ THEN
                IF statDirectParameter1 THEN

                    data^.directParameterPage.masterCommand       :=    statRecord[0];
                    data^.directParameterPage.masterCycleTime     :=    statRecord[1];
                    data^.directParameterPage.minCycleTime        :=    statRecord[2];
                    data^.directParameterPage.frameCapability     :=    statRecord[3];
                    data^.directParameterPage.ioLinkRevisionID    :=    statRecord[4];
                    data^.directParameterPage.processDataIn       :=    statRecord[5];
                    data^.directParameterPage.processDataOut      :=    statRecord[6];
                    data^.directParameterPage.vendorID1           :=    statRecord[7];
                    data^.directParameterPage.vendorID2           :=    statRecord[8];
                    data^.directParameterPage.deviceID1           :=    statRecord[9];
                    data^.directParameterPage.deviceID2           :=    statRecord[10];
                    data^.directParameterPage.deviceID3           :=    statRecord[11];
                    data^.directParameterPage.functionID1         :=    statRecord[12];
                    data^.directParameterPage.functionID2         :=    statRecord[13];
                    data^.directParameterPage.reserved1           :=    statRecord[14];
                    data^.directParameterPage.reserved2           :=    statRecord[15];

                ELSIF statDeviceAccessLocks THEN
                    data^.deviceAccessLocks.%B0 := statRecord[0];
                    data^.deviceAccessLocks.%B1 := statRecord[1];

                ELSIF statVendorName THEN
                    tempData256[0]  := TO_BYTE(statRecordLen);
                    FOR tempIndex := UINT#0 TO TO_UINT(statRecordLen) - UINT#0 DO
                        tempData256[tempIndex + UINT#1] := statRecord[tempIndex];
                    END_FOR;
                    Deserialize(UINT#0,tempData256,data^.vendorName);
                ELSIF statVendorText THEN
                    tempData256[0]  := TO_BYTE(statRecordLen);
                    FOR tempIndex := UINT#0 TO TO_UINT(statRecordLen) - UINT#0 DO
                        tempData256[tempIndex + UINT#1] := statRecord[tempIndex];
                    END_FOR;
                    Deserialize(UINT#0,tempData256,data^.vendorText);

                ELSIF statProductName THEN
                    tempData256[0]  := TO_BYTE(statRecordLen);
                    FOR tempIndex := UINT#0 TO TO_UINT(statRecordLen) - UINT#0 DO
                        tempData256[tempIndex + UINT#1] := statRecord[tempIndex];
                    END_FOR;
                    Deserialize(UINT#0,tempData256,data^.productName);

                ELSIF statProductID THEN
                    tempData256[0]  := TO_BYTE(statRecordLen);
                    FOR tempIndex := UINT#0 TO TO_UINT(statRecordLen) - UINT#0 DO
                        tempData256[tempIndex + UINT#1] := statRecord[tempIndex];
                    END_FOR;
                    Deserialize(UINT#0,tempData256,data^.productID);

                ELSIF statProductText THEN
                    tempData256[0]  := TO_BYTE(statRecordLen);
                    FOR tempIndex := UINT#0 TO TO_UINT(statRecordLen) - UINT#0 DO
                        tempData256[tempIndex + UINT#1] := statRecord[tempIndex];
                    END_FOR;
                    Deserialize(UINT#0,tempData256,data^.productText);

                ELSIF statSerialNumber THEN
                    FOR tempIndex := UINT#0 TO TO_UINT(statRecordLen) - UINT#0 DO
                        tempData256[tempIndex + UINT#1] := statRecord[tempIndex];
                    END_FOR;
                    Deserialize(UINT#0,tempData256,data^.serialNumber);

                ELSIF statHwRevision THEN
                    tempData256[0]  := TO_BYTE(statRecordLen);
                    FOR tempIndex := UINT#0 TO TO_UINT(statRecordLen) - UINT#0 DO
                        tempData256[tempIndex + UINT#1] := statRecord[tempIndex];
                    END_FOR;
                    Deserialize(UINT#0,tempData256,data^.hwRevision);

                ELSIF statFwRevision THEN
                    tempData256[0]  := TO_BYTE(statRecordLen);
                    FOR tempIndex := UINT#0 TO TO_UINT(statRecordLen) - UINT#0 DO
                        tempData256[tempIndex + UINT#1] := statRecord[tempIndex];
                    END_FOR;
                    Deserialize(UINT#0,tempData256,data^.fwRevision);

                ELSIF statAppSpecificName THEN
                    tempData256[0]  := TO_BYTE(statRecordLen);
                    FOR tempIndex := UINT#0 TO TO_UINT(statRecordLen) - UINT#0 DO
                        tempData256[tempIndex + UINT#1] := statRecord[tempIndex];
                    END_FOR;
                    Deserialize(UINT#0,tempData256,data^.appSpecificName);

                ELSIF statErrorCount THEN
                    data^.errorCount.%B0 := statRecord[1];
                    data^.errorCount.%B1 := statRecord[0];

                ELSIF statDeviceStatus THEN
                    data^.deviceStatus := statRecord[0];

                ELSIF statDeviceStatusDetailed THEN
                    data^.deviceStatusDetailed := statRecord[0];

                ELSIF statProcessIn THEN
                    FOR tempIndex := UINT#0 TO TO_UINT(statRecordLen) - UINT#1 DO
                        data^.processImageIn[tempIndex] :=  statRecord[tempIndex];
                    END_FOR;

                ELSIF statProcessOut THEN
                    FOR tempIndex := UINT#0 TO TO_UINT(statRecordLen) - UINT#1 DO
                        data^.processImageOut[tempIndex] :=  statRecord[tempIndex];
                    END_FOR;

                ELSIF statParameters THEN
                    data^.parameters.eventMessage    := statRecord[0];
                    data^.parameters.operatingMode   := statRecord[1];
                    data^.parameters.readyDelay      := statRecord[2];
                    data^.parameters.dataHoldingTime := statRecord[3];
                    data^.parameters.rfParameters    := statRecord[4];
                    data^.parameters.modulation      := statRecord[5];
                    data^.parameters.subcarrier      := statRecord[6];
                    data^.parameters.dataTransfer    := statRecord[7];

                ELSIF statEventHistory THEN
                    data^.eventHistory.lastEvent.%B0                :=	statRecord[3];
                    data^.eventHistory.lastEvent.%B1                :=	statRecord[2];
                    data^.eventHistory.lastEvent.%B2                :=	statRecord[1];
                    data^.eventHistory.lastEvent.%B3                :=	statRecord[0];

                    data^.eventHistory.secondLastEvent.%B0          :=	statRecord[7];
                    data^.eventHistory.secondLastEvent.%B1          :=	statRecord[6];
                    data^.eventHistory.secondLastEvent.%B2          :=	statRecord[5];
                    data^.eventHistory.secondLastEvent.%B3          :=	statRecord[4];

                    data^.eventHistory.thirdLastEvent.%B0           :=	statRecord[11];
                    data^.eventHistory.thirdLastEvent.%B1           :=	statRecord[10];
                    data^.eventHistory.thirdLastEvent.%B2           :=	statRecord[9];
                    data^.eventHistory.thirdLastEvent.%B3           :=	statRecord[8];

                    data^.eventHistory.fourthLastEvent.%B0          :=	statRecord[15];
                    data^.eventHistory.fourthLastEvent.%B1          :=	statRecord[14];
                    data^.eventHistory.fourthLastEvent.%B2          :=	statRecord[13];
                    data^.eventHistory.fourthLastEvent.%B3          :=	statRecord[12];

                    data^.eventHistory.fifthLastEvent.%B0           :=	statRecord[19];
                    data^.eventHistory.fifthLastEvent.%B1           :=	statRecord[18];
                    data^.eventHistory.fifthLastEvent.%B2           :=	statRecord[17];
                    data^.eventHistory.fifthLastEvent.%B3           :=	statRecord[16];

                ELSIF statReaderStatus THEN
                    data^.readerStatus.timeSinceStartup.%B0         :=  statRecord[3];
                    data^.readerStatus.timeSinceStartup.%B1         :=  statRecord[2];
                    data^.readerStatus.timeSinceStartup.%B2         :=  statRecord[1];
                    data^.readerStatus.timeSinceStartup.%B3         :=  statRecord[0];
                    data^.readerStatus.tagsInTheField               :=	statRecord[4];
                    data^.readerStatus.antennaStatus                :=  statRecord[5];
                    data^.readerStatus.tagChanges.%B0               :=  statRecord[9];
                    data^.readerStatus.tagChanges.%B1               :=  statRecord[8];
                    data^.readerStatus.tagChanges.%B2               :=  statRecord[7];
                    data^.readerStatus.tagChanges.%B3               :=  statRecord[6];
                    data^.readerStatus.lineDriverRev                :=  statRecord[10];
                    data^.readerStatus.errorCounterPassive          :=  statRecord[11];
                    data^.readerStatus.abortCounter                 :=  statRecord[12];
                    data^.readerStatus.codeErrorCounter             :=  statRecord[13];
                    data^.readerStatus.signatureErrorCounter        :=  statRecord[14];
                    data^.readerStatus.crcErrorCounter              :=  statRecord[15];
                    data^.readerStatus.currentCommandStatus         :=  statRecord[16];
                    data^.readerStatus.errorCount                   :=  statRecord[17];

                ELSIF statTagStatus THEN
                    data^.tagStatus.uid[0]              :=  statRecord[0];
                    data^.tagStatus.uid[1]              :=  statRecord[1];
                    data^.tagStatus.uid[2]              :=  statRecord[2];
                    data^.tagStatus.uid[3]              :=  statRecord[3];
                    data^.tagStatus.uid[4]              :=  statRecord[4];
                    data^.tagStatus.uid[5]              :=  statRecord[5];
                    data^.tagStatus.uid[6]              :=  statRecord[6];
                    data^.tagStatus.uid[7]              :=  statRecord[7];
                    data^.tagStatus.tagName             :=  statRecord[8];
                    data^.tagStatus.chipVersion         :=  statRecord[9];
                    data^.tagStatus.memSize.%B0         :=  statRecord[11];
                    data^.tagStatus.memSize.%B1         :=  statRecord[10];
                    data^.tagStatus.lockStatus          :=  statRecord[12];
                    data^.tagStatus.memBlockSize        :=  statRecord[13];
                    data^.tagStatus.numBlocks           :=  statRecord[14];

                ELSIF statUidHistory THEN
                    data^.uidHistory.lastUID1.%B0         :=  statRecord[3];
                    data^.uidHistory.lastUID1.%B1         :=  statRecord[2];
                    data^.uidHistory.lastUID1.%B2         :=  statRecord[1];
                    data^.uidHistory.lastUID1.%B3         :=  statRecord[0];
                    data^.uidHistory.lastUID2.%B0         :=  statRecord[7];
                    data^.uidHistory.lastUID2.%B1         :=  statRecord[6];
                    data^.uidHistory.lastUID2.%B2         :=  statRecord[5];
                    data^.uidHistory.lastUID2.%B3         :=  statRecord[4];
                    data^.uidHistory.secondLastUID1.%B0   :=  statRecord[11];
                    data^.uidHistory.secondLastUID1.%B1   :=  statRecord[10];
                    data^.uidHistory.secondLastUID1.%B2   :=  statRecord[9];
                    data^.uidHistory.secondLastUID1.%B3   :=  statRecord[8];
                    data^.uidHistory.secondLastUID2.%B0   :=  statRecord[15];
                    data^.uidHistory.secondLastUID2.%B1   :=  statRecord[14];
                    data^.uidHistory.secondLastUID2.%B2   :=  statRecord[13];
                    data^.uidHistory.secondLastUID2.%B3   :=  statRecord[12];
                    data^.uidHistory.thirdLastUID1.%B0    :=  statRecord[19];
                    data^.uidHistory.thirdLastUID1.%B1    :=  statRecord[18];
                    data^.uidHistory.thirdLastUID1.%B2    :=  statRecord[17];
                    data^.uidHistory.thirdLastUID1.%B3    :=  statRecord[16];
                    data^.uidHistory.thirdLastUID2.%B0    :=  statRecord[23];
                    data^.uidHistory.thirdLastUID2.%B1    :=  statRecord[22];
                    data^.uidHistory.thirdLastUID2.%B2    :=  statRecord[21];
                    data^.uidHistory.thirdLastUID2.%B3    :=  statRecord[20];
                    data^.uidHistory.fourthLastUID1.%B0   :=  statRecord[27];
                    data^.uidHistory.fourthLastUID1.%B1   :=  statRecord[26];
                    data^.uidHistory.fourthLastUID1.%B2   :=  statRecord[25];
                    data^.uidHistory.fourthLastUID1.%B3   :=  statRecord[24];
                    data^.uidHistory.fourthLastUID2.%B0   :=  statRecord[31];
                    data^.uidHistory.fourthLastUID2.%B1   :=  statRecord[30];
                    data^.uidHistory.fourthLastUID2.%B2   :=  statRecord[29];
                    data^.uidHistory.fourthLastUID2.%B3   :=  statRecord[28];
                    data^.uidHistory.fifthLastUID1.%B0    :=  statRecord[35];
                    data^.uidHistory.fifthLastUID1.%B1    :=  statRecord[34];
                    data^.uidHistory.fifthLastUID1.%B2    :=  statRecord[33];
                    data^.uidHistory.fifthLastUID1.%B3    :=  statRecord[32];
                    data^.uidHistory.fifthLastUID2.%B0    :=  statRecord[39];
                    data^.uidHistory.fifthLastUID2.%B1    :=  statRecord[38];
                    data^.uidHistory.fifthLastUID2.%B2    :=  statRecord[37];
                    data^.uidHistory.fifthLastUID2.%B3    :=  statRecord[36];

                ELSE // Other data sets are not defined
                    ;
                END_IF;
                tempInternalError := tempRetValDeserialize <> TO_INT(STATUS_EXECUTION_FINISHED);
            END_IF;

            statDoneOld := instDevice_done;

            // OUTPUTS
            IF tempInternalError THEN //Error occured
                done := false;
                busy := false;
                error := true;
                status := ERR_INCONSISTENT_DATA;
            ELSE //Execute successful
                done := instDevice_done;
                busy := instDevice_busy;
                error := instDevice_error;
                status := instDevice_status;
                diagnostics^ := instDevice_diagnostics;
            END_IF;
        END_METHOD
    END_CLASS
END_NAMESPACE

(* ---- AxoIOLink_RF200_ReadTag.st ---- *)
USING AXOpen.Components.Abstractions.Drives;
USING AXOpen.Timers;
USING Siemens.Simatic.S71500.DistributedIO;
USING System.Timer;
USING System.Strings;
USING System.Serialization;

NAMESPACE AXOpen.Components.SIEM.Identification
    {S7.extern=ReadWrite}
    CLASS PUBLIC AxoIOLink_RF200_ReadTag
        VAR PRIVATE
            statPae                 :	ARRAY[0..UPPER_BOUND_NETTO_IO_FIELD] OF BYTE;       //  Partly recived identification data vie Process image
            statStatusByte          :	BYTE    :=  BYTE#0;                                 //  RF200 Tag reader status byte
            statPresence            :	BOOL    :=  FALSE;                                  //  TRUE: Transponder on field
            statState               :	INT     :=  INT#0;	                                //  Main State Machine Index
            statAddr                :	WORD    :=  WORD#0;                                 //  Start address of data on tag
            statOffset              :	INT     :=  INT#0;	                                //  Buffer offset
            statExecuteReq          :	BOOL    :=  FALSE;                                  //  Execute function memory
            statLength              :	DINT    :=  DINT#0;	                                //  Length of read data
            statDat                 :	ARRAY[0..UPPER_BOUND_IO_FIELD] OF BYTE;             //	Data to Send
            statRecDat              :	ARRAY[0..UPPER_BOUND_IO_FIELD] OF BYTE;             //	Data Received
            statAddrOffset          :	INT     :=  INT#0;	                                //  Start adress of port
            statPresenceFF          :	BOOL    :=  FALSE;                                  //  TRUE: Transponder on field
            instTonrTime            :	TimeAccumulator;                                    //  Tag has left antenna field detection timer
            statTimerIn             :	BOOL    :=  FALSE;                                  //  Tag has left antenna field detection timer - Start Tag
            statTimerR              :	BOOL    :=  FALSE;                                  //  Tag has left antenna field detection timer - Reset Tag
            statTimerPt             :	TIME	:=  DETECTION_TIME_TAG_OFF_FIELD;           //  Tag has left antenna field detection timer - Detection time
            statReadData            :	ARRAY[0..UPPER_BOUND_MAX_DATA_FIELD] OF BYTE;		//  Received tag identification data
            statCountCopyPae        :	DINT    :=  DINT#0;	                                //  Length of current next data part in process image
            statBusy                :	BOOL    :=  FALSE;                                  //  TRUE: FB is not finished and new output values can be expected
            statDone                :	BOOL    :=  FALSE;                                  //  TRUE: Commanded functionality has been completed successfully
            statError               :	BOOL    :=  FALSE;                                  //  TRUE: Commanded functionality has been canceled with error
            statReturnMoveBlkVar    :	INT     :=  INT#0;	                                //  Return Value PAE copy function
            statDiffToIOsizeNetto   :	INT     :=  INT#0;	                                //  Difference between requested length and PAE
            statIoPartError         :	BOOL    :=  FALSE;                                  //  TRUE: data in process image is invalid
            statIoPartStatus        :	DWORD   :=  DWORD#0;                                //  Status for IO access
            statIOsize              :	USINT   :=  USINT#0;	                            //  Size of the IO-Link Master PII
            statIOsizeNetto         :	USINT   :=  USINT#0;	                            //  Size of the IO-Link Master PAE without header
            statIdentDataLowIndex   :   INT     :=  INT#0;
            statIdentDataHighIndex  :   INT     :=  INT#0;
        END_VAR

        VAR CONSTANT
            IOL_V10                         :	USINT   :=  USINT#10;       //  Identifier IO-Link version 1.0
            IOL_V11                         :	USINT   :=  USINT#11;       //  Identifier IO-Link version 1.1
            LEN_DATA_V10                    :	USINT   :=  USINT#8;        //  Length of user data for IO-Link version 1.0
            LEN_DATA_V11                    :	USINT   :=  USINT#32;       //  Length of user data for IO-Link version 1.1
            UPPER_BOUND_IO_FIELD            :	USINT   :=  USINT#31;       //  Upper bound of Input and Output fields
            UPPER_BOUND_NETTO_IO_FIELD      :	USINT   :=  USINT#27;       //  Upper bound of Input and Output fields without header
            UPPER_BOUND_MAX_DATA_FIELD      :	UINT    :=  UINT#1999;      //  Upper bound of the data field of a RFID Tag
            DATA_HEADER_SIZE                :	USINT   :=  USINT#4;        //  IO-Link Header Size for version 1.0 and 1.1
            CMD_READ                        :	BYTE    :=  BYTE#16#02;     //  Command to read data
            CMD_RESET                       :	BYTE    :=  BYTE#16#00;     //  Command to reset
            MIN_LENGTH_V10                  :	WORD    :=  WORD#16#0004;   //  Minimal Lenght of requested tag information
            MIN_LENGTH_V11                  :	WORD    :=  WORD#16#001C;   //  Minimal Lenght of requested tag information
            STATUS_ERROR_IDENT_BLOCK        :	WORD    :=  WORD#16#0001;   //  Error Identification for block internal faults
            STATUS_ERROR_IDENT_RFID         :	WORD    :=  WORD#16#0011;   //  Error Identification for RFID reader faults
            STATUS_NO_JOB                   :	WORD    :=  WORD#16#0000;   //  No job requested
            STATUS_ERROR_TAG_HAS_LEFT       :	WORD    :=  WORD#16#8101;   //  Error - the RFID tag has left the reader
            STATUS_ERROR_STILL_ACTIVE       :	WORD    :=  WORD#16#8102;   //  Error - block still busy, no further request possible
            STATUS_ERROR_LENGTH             :	WORD    :=  WORD#16#8104;   //  Error - requested length is less than 0
            STATE_IDLE                      :	INT     :=  INT#0;          //  State Machine - Idle State
            STATE_READ                      :	INT     :=  INT#2;          //  State Machine - Read Tag
            STATE_TELEGRAM                  :	INT     :=  INT#1;          //  State Machine - Prepare telegram
            STATE_ERROR                     :	INT     :=  INT#3;          //  State Machine - Error State
            DETECTION_TIME_TAG_OFF_FIELD    :	TIME    :=  T#5S;           //  Tag has left antenna field detection time
            INDEX_CMD                       :	USINT   :=  USINT#0;        //  Index in DataField - Command
            INDEX_RFID_ERROR                :	USINT   :=  USINT#1;        //  Index in DataField - Error
            INDEX_ADDR_HIGH                 :	USINT   :=  USINT#2;        //  Index in DataField - Address High Byte
            INDEX_ADDR_LOW                  :	USINT   :=  USINT#3;        //  Index in DataField - Address Low Byte
            INDEX_SOURCE_DATA               :	DINT    :=  DINT#4;         //  Index in Data Field - Start of netto Data

        END_VAR

        METHOD PUBLIC Run
            VAR_INPUT
                execute     :	BOOL    :=  FALSE;          //  Request job (on rising edge)
                addrTag     :	WORD    :=  WORD#16#0;      //  Start address of data on tag
                length      :	WORD    :=  WORD#16#0;      //	Length of data to be read
                hwID        :	WORD    :=  WORD#16#0;      //	Logic IO address of the IO-Link Master
                portAddr    :	INT     :=  INT#0;          //  Start address of port
                version     :	USINT   :=  IOL_V11;        //	IO-Link version of the reader; 11: IO-Link V1.1, 10: IO-Link V1.0
                identData   :   REF_TO  ARRAY[*]OF BYTE;    //  Received tag identification data
            END_VAR

            VAR_OUTPUT
                done        :	BOOL;       //  FALSE: data invalid, TRUE: data valid
                busy        :	BOOL;       //  FALSE: no job, TRUE: job in progress
                error       :	BOOL;       //  FALSE: no error, TRUE: error
                status      :	DWORD;      //  Error status
                presence    :	BOOL;       //  TRUE: Transponder on field
            END_VAR

            VAR_TEMP
                tempStatus  :   DWORD;  //  Auxiliary tag for status output
                tempWord    :   WORD;
                tempIndex   :   INT;
                tempHWData  :   ARRAY[0..255] OF BYTE;
            END_VAR

            IF identData = NULL THEN
                // TODO some message
                error := TRUE;
                status  := DWORD#16#FEFE0001;
                RETURN;
            END_IF;

            statIdentDataLowIndex := TO_INT(LOWER_BOUND(identData^, 1));
            statIdentDataHighIndex := TO_INT(UPPER_BOUND(identData^, 1));

            // INFO HEADER
            //===============================================================================
            // Siemens / (c)Copyright 2022
            //-------------------------------------------------------------------------------
            // Title:            LIOLink_RF200_ReadTag
            // Function:         Reads tags from SIMATIC RF200 readers via IO-Link
            // Library:          LIOLink
            // Author:           Siemens Industry Online Support
            // Tested with:      CPU 1513-1 PN FW 2.8
            // Engineering:      TIA Portal V16
            // Restrictions:     --
            // Requirements:     --
            //-------------------------------------------------------------------------------
            // Change log table:
            // Version  | Date       | Expert in charge       | Changes applied
            //----------|------------|------------------------|------------------------------
            // 01.00.00 | 01.07.2013 | Online Support         | First release
            // 01.01.00 | 01.12.2016 | Online Support         | Upgraded to TIA Portal V14
            // 02.00.00 | 01.09.2017 | Online Support         | Upgraded to TIA Portal V14 SP1
            //                                                | Implemented Programming styleguide
            //                                                | Added support for IO-Link V1.1 readers
            // 02.01.00 | 01.12.2017 | Online Support         | Bug fixes and performance improvements
            // 02.02.00 | 01.03.2020 | Online Support         | Upgraded to TIA Portal V16
            // 02.03.00 | 22.09.2020 | Online Support         | Integrated FB into LIOLink library
            //                                                | Renamed FB to LIOLink_RF200_ReadTag
            //                                                | Combined FBs for IO-Link V1.0 and V1.1
            //                                                | Minor bug fixes
            // 02.04.00 | 29.06.2022 | Online Support         | Minor bug fixes
            // 02.05.00 | 30.09.2022 | SUP SPH                | Optimization
            //===============================================================================

            // Check version
            //determine IO-Link reader version (1.0/1.1) to set offsets
            IF version = IOL_V11 THEN
                statIOsize := LEN_DATA_V11;
                statIOsizeNetto := LEN_DATA_V11 - DATA_HEADER_SIZE;
            ELSE
                statIOsize := LEN_DATA_V10;
                statIOsizeNetto := LEN_DATA_V10 - DATA_HEADER_SIZE;
            END_IF;

            // Get PII
            statAddrOffset := portAddr;   //start adress of port

            // Read PII
            tempWord := Siemens.Simatic.S71500.DistributedIO.ReadData(hwID,tempHWData);
            statIoPartStatus := tempWord;
            statIoPartError := tempWord > WORD#0;

            FOR tempIndex := 0 TO statIOsize - INT#1 DO
                statRecDat[tempIndex]   :=  tempHWData[tempIndex + statAddrOffset];
            END_FOR;

            statStatusByte := statRecDat[0];    //Status Byte
            statPresence := statStatusByte.%X5;   //Presence bit. Transponder on field

            // Check execute
            // Idle
                IF NOT execute THEN
                    statDone    :=  false;
                    statBusy    :=  false;
                    statError   :=  false;
                    tempStatus  :=  STATUS_NO_JOB;
                END_IF;

            // Job requested
                //Positive edge for reading of data
                IF execute AND execute <> statExecuteReq THEN
                    IF NOT statBusy THEN
                        statAddr := addrTag;    //Transpoder Address
                        statDiffToIOsizeNetto := TO_INT(length) MOD statIOsizeNetto;
                        statLength := TO_DINT(length);   //Length of read Dat
                        statBusy := TRUE;
                        statDone := FALSE;
                        statError := FALSE;
                        tempStatus := STATUS_NO_JOB;
                        statOffset := 0;   //offset of puffer must be reseted
                        statState := STATE_READ;    //next step >> send read command
                        statCountCopyPae := 0;

                        FOR tempIndex := statIdentDataLowIndex TO statIdentDataHighIndex DO
                            identData^[tempIndex] := BYTE#0;
                        END_FOR;
                    ELSE
                        tempStatus.%W0 := STATUS_ERROR_STILL_ACTIVE;                       //block is still active
                        tempStatus.%W1 := STATUS_ERROR_IDENT_BLOCK;                        //Error identifier for block errors
                        statState := STATE_ERROR;
                    END_IF;
                    IF length < WORD#0 OR (length < MIN_LENGTH_V11 AND version = IOL_V11) OR (length < MIN_LENGTH_V10 AND version = IOL_V10) THEN
                        tempStatus.%W0 := STATUS_ERROR_LENGTH;                             //length too short
                        tempStatus.%W1 := STATUS_ERROR_IDENT_BLOCK;                        //identifier rfid errors
                        statState := STATE_ERROR;
                    END_IF;
                END_IF;
            statExecuteReq := execute;

        // Tag presence detection
            IF NOT statPresence AND statPresence <> statPresenceFF THEN   //the tag has left the antenna  field
                IF NOT statDone THEN
                    statTimerIn := true;   //wait 5 sec
                    statTimerR := false;
                END_IF;
            END_IF;
            statPresenceFF := statPresence;
            IF statPresence THEN
                statTimerR := true;
                statTimerIn := false;
            END_IF;

        // State machine
            CASE statState OF
                STATE_IDLE:
                    statBusy := false;
                    statTimerIn := false;

                STATE_READ:
                    IF statLength > 0 THEN
                        statDat[INDEX_CMD] := CMD_READ;    //Set read command
                        statDat[INDEX_ADDR_HIGH] := statAddr.%B1;    //Adr-H
                        statDat[INDEX_ADDR_LOW] := statAddr.%B0;   //Adr-L
                    END_IF;

                    IF NOT statIoPartError THEN
                        statState := STATE_TELEGRAM;    //Telegram: Edit the read data
                    END_IF;

                STATE_TELEGRAM:
                    IF statLength > 0 THEN   //Only when length of data>0 can continue
                        IF statStatusByte.%X6 THEN   //IF RFID error has occured
                            tempStatus.%W0 := statRecDat[INDEX_RFID_ERROR];    //error_RFID
                            tempStatus.%W1 := STATUS_ERROR_IDENT_RFID;    //Error identifier for RFID errors
                            statState := STATE_ERROR;
                        END_IF;

                        //-------------------------- read command is ready------------------------------------------------//
                        IF statStatusByte.%X7 AND statStatusByte.%X1 THEN
                            IF statRecDat[INDEX_ADDR_HIGH] = statAddr.%B1
                                AND statRecDat[INDEX_ADDR_LOW] = statAddr.%B0
                            THEN //received ADR must be ==sent ADR

                                FOR tempIndex := INT#0 TO TO_INT(statIOsizeNetto) - INT#1 DO
                                    statPae[tempIndex]  :=  statRecDat[tempIndex + INDEX_SOURCE_DATA];
                                END_FOR;

                                IF NOT statIoPartError THEN
                                    IF statCountCopyPae = 0 THEN    //copy the statIOsizeNet Bytes in
                                        IF statLength >= statIOsizeNetto THEN
                                            IF statLength <> TO_DINT(length) THEN
                                                statAddr := TO_WORD(TO_INT(statAddr) + statIOsizeNetto);
                                            END_IF;
                                            statState := STATE_READ;
                                            statCountCopyPae := statIOsizeNetto;
                                        ELSE
                                            IF statStatusByte.%X7 AND NOT statStatusByte.%X6 THEN
                                                IF statDiffToIOsizeNetto <> 0 THEN
                                                    statCountCopyPae := statDiffToIOsizeNetto;
                                                    statAddr := TO_WORD(TO_INT(statAddr) + statIOsizeNetto);
                                                    statState := STATE_READ;
                                                ELSE
                                                    statCountCopyPae := statIOsizeNetto;
                                                END_IF;
                                            ELSE
                                                statState := STATE_IDLE;
                                            END_IF;
                                        END_IF;
                                    ELSE
                                        FOR tempIndex := INT#0 TO TO_INT(statCountCopyPae) - INT#1 DO
                                            statReadData[tempIndex + statOffset]  :=  statPae[tempIndex];
                                        END_FOR;

                                        IF statReturnMoveBlkVar = 0 THEN
                                            statCountCopyPae := 0;
                                            statOffset := statOffset + statIOsizeNetto;
                                            statLength := statLength - statIOsizeNetto;
                                        END_IF;
                                    END_IF;
                                ELSE
                                    tempStatus.%W0 := TO_WORD(statIoPartStatus); //Error has to BLKMOV occured
                                    tempStatus.%W1 := STATUS_ERROR_IDENT_BLOCK;   //functions-Error identifier
                                    statState := STATE_ERROR;
                                END_IF;
                            END_IF;
                        END_IF;

                        FOR tempIndex := INT#0 TO statIOsize - INT#1 DO
                            tempHWData[tempIndex + statAddrOffset] := statDat[tempIndex];
                        END_FOR;
                        //TODO solve overwriting the outputs in case of several RFID header used with one IOLink master
                        //when SETIO_PART equivalent function is available in AX
                        tempWord := Siemens.Simatic.S71500.DistributedIO.WriteData(hwID,tempHWData);
                        statIoPartStatus := tempWord;
                        statIoPartError := tempWord > WORD#0;

                        IF statIoPartError THEN
                            tempStatus.%W0 := TO_WORD(statIoPartStatus);    //Error has to BLKMOV occured
                            tempStatus.%W1 := STATUS_ERROR_IDENT_BLOCK;   //functions-Error identifier
                            statState := STATE_ERROR;
                        END_IF;

                    ELSE

                        FOR tempIndex := INT#0 TO statIdentDataHighIndex - statIdentDataLowIndex - INT#1 DO
                            identData^[tempIndex + statIdentDataLowIndex]  :=  statReadData[tempIndex];
                        END_FOR;

                        statState := STATE_IDLE;
                        statBusy := false;
                        statDone := true;

                        //Reset read command
                        statDat[INDEX_CMD] := CMD_RESET;

                        FOR tempIndex := INT#0 TO statIOsize - INT#1 DO
                            tempHWData[tempIndex + statAddrOffset] := statDat[tempIndex];
                        END_FOR;
                        //TODO solve overwriting the outputs in case of several RFID header used with one IOLink master
                        //when SETIO_PART equivalent function is available in AX
                        tempWord := Siemens.Simatic.S71500.DistributedIO.WriteData(hwID,tempHWData);
                        statIoPartStatus := tempWord;
                        statIoPartError := tempWord > WORD#0;
                    END_IF;

                STATE_ERROR:
                    statBusy := false;
                    statDone := false;
                    statError := true;
                    statTimerIn := false;
                    statTimerR := true;
                    statState := STATE_IDLE;

                    //Reset read command
                    statDat[INDEX_CMD] := CMD_RESET;

                    FOR tempIndex := INT#0 TO statIOsize - INT#1 DO
                        tempHWData[tempIndex + statAddrOffset] := statDat[tempIndex];
                    END_FOR;
                    //TODO solve overwriting the outputs in case of several RFID header used with one IOLink master
                    //when SETIO_PART equivalent function is available in AX
                    tempWord := Siemens.Simatic.S71500.DistributedIO.WriteData(hwID,tempHWData);
                    statIoPartStatus := tempWord;
                    statIoPartError := tempWord > WORD#0;
                ELSE
                    statState := STATE_IDLE;
            END_CASE;

            // Detection timer
            instTonrTime(signal := statTimerIn,   //this timer will start, if the tag has left the antenna field
                          reset := statTimerR,
                          duration := statTimerPt);
            IF instTonrTime.output THEN   //error has occured. No tag on field during the 5 sec.
                tempStatus.%W0 := STATUS_ERROR_TAG_HAS_LEFT;    //tag has left the field
                tempStatus.%W1 := STATUS_ERROR_IDENT_BLOCK;   //identifier rfid errors
                statState := STATE_ERROR;
            END_IF;

            // Update output interface
            done := statDone;
            busy := statBusy;
            error := statError;
            status := tempStatus;
            presence := statPresence;
        END_METHOD
    END_CLASS
END_NAMESPACE
